// TwinCAT 3 PLC project pruebaPaletizada
// ProgramVersion: 3.1.4024.0
// libraries:
//   Tc2_Standard, * (Beckhoff Automation GmbH)
//   Tc2_System, * (Beckhoff Automation GmbH)
//   Tc3_Module, * (Beckhoff Automation GmbH)
//   VisuSymbols,3.5.10.0,System
// project tree:
//   / GlobalTextList.TcGTLO, PlcTask.TcTTO, Visualization Manager.TcVMO (not stored)
//   GVLs/ GVLvars.TcGVL
//   POUs/ MAIN.TcPOU
//   VISUs/ HMI.TcVIS
// real-time tasks:
//   TASK PlcTask: cycle T#10ms, priority 20, ADS port 350

CONFIGURATION pruebaPaletizada
    RESOURCE PLC ON TwinCAT3
        TASK PlcTask(INTERVAL := T#10ms, PRIORITY := 20);
        PROGRAM MAIN WITH PlcTask : MAIN;
    END_RESOURCE
END_CONFIGURATION

// ---- GVLs/GVLvars.TcGVL
{attribute 'qualified_only'}
VAR_GLOBAL
	// Cuadro
	{attribute 'OPC.UA.DA' := '1'}
	botonStart : BOOL;
	{attribute 'OPC.UA.DA' := '1'}
	botonStop : BOOL;
	{attribute 'OPC.UA.DA' := '1'}
	seta : BOOL; 
	{attribute 'OPC.UA.DA' := '1'}
	botonReset : BOOL;
	{attribute 'OPC.UA.DA' := '1'}
	luzStart : BOOL;
	{attribute 'OPC.UA.DA' := '1'}
	luzStop : BOOL;
	{attribute 'OPC.UA.DA' := '1'}
	luzReset : BOOL;
	{attribute 'OPC.UA.DA' := '1'}
	luzVerde : BOOL;
	{attribute 'OPC.UA.DA' := '1'}
	luzRoja : BOOL;
	{attribute 'OPC.UA.DA' := '1'}
	luzAmarilla : BOOL;
	
	
	// Sensores 
	{attribute 'OPC.UA.DA' := '1'}
	sDifusoCintaMaterial : BOOL;
	{attribute 'OPC.UA.DA' := '1'}
	sEntradaPaletizadorMaterial : BOOL;
	{attribute 'OPC.UA.DA' := '1'}
	sEntradaMesaRotation : BOOL;
	{attribute 'OPC.UA.DA' := '1'}
	sSalidaMesaRotacion : BOOL;
	{attribute 'OPC.UA.DA' := '1'}
	sPostPaletizado : BOOL;
	{attribute 'OPC.UA.DA' := '1'}
	sEntradaPaletEnEstacion : BOOL;
	{attribute 'OPC.UA.DA' := '1'}
	sBasePalet : BOOL ;
	{attribute 'OPC.UA.DA' := '1'}
	numProductosCompletos : INT;
	
	

	// Cintas
	{attribute 'OPC.UA.DA' := '1'}
	cintaEntradaMaterial : BOOL;
	{attribute 'OPC.UA.DA' := '1'}
	cintaInclinadaMaterial : BOOL;
	{attribute 'OPC.UA.DA' := '1'}
	cintaEntradaPalets : BOOL;
	{attribute 'OPC.UA.DA' := '1'}
	cintaSalida : BOOL;
	{attribute 'OPC.UA.DA' := '1'}
	cintaPaletEntradaEstacion : BOOL;
	
	// Mesa Giratoria (Monoestable)
	// Output
	{attribute 'OPC.UA.DA' := '1'}
	turnMesaGiratoria : BOOL;
	{attribute 'OPC.UA.DA' := '1'}
	load : BOOL;
	{attribute 'OPC.UA.DA' := '1'}
	unload : BOOL;
	// Input
	{attribute 'OPC.UA.DA' := '1'}
	frontLimit : BOOL; // Limite frontal de la mesa giratoria
	{attribute 'OPC.UA.DA' := '1'}
	backLimit : BOOL; // Limite trasero de la mesa giratoria
	{attribute 'OPC.UA.DA' := '1'}
	minuminRotation : BOOL; // rotation limit 0
	{attribute 'OPC.UA.DA' := '1'}
	maximunRotation : BOOL; // rotation limit 90
	
	// Paletizador Salidas
	{attribute 'OPC.UA.DA' := '1'}
	pusher : BOOL;
	{attribute 'OPC.UA.DA' := '1'}
	turnFlipper : BOOL;
	{attribute 'OPC.UA.DA' := '1'}
	moveClamper : BOOL;
	{attribute 'OPC.UA.DA' := '1'}
	beltPositive : BOOL;
	{attribute 'OPC.UA.DA' := '1'}
	beltNegative : BOOL;
	{attribute 'OPC.UA.DA' := '1'}
	chainPositive : BOOL;
	{attribute 'OPC.UA.DA' := '1'}
	chainNegative : BOOL;
	{attribute 'OPC.UA.DA' := '1'}
	OpenPlate : BOOL;
	{attribute 'OPC.UA.DA' := '1'}
	elevatorUp : BOOL;
	{attribute 'OPC.UA.DA' := '1'}
	elevatorDown : BOOL;
	{attribute 'OPC.UA.DA' := '1'}
	elevatorToLimit : BOOL;
	
	
	// Paletizador Entradas
	{attribute 'OPC.UA.DA' := '1'}
	clamped : BOOL;
	{attribute 'OPC.UA.DA' := '1'}
	plateLimit : BOOL;
	{attribute 'OPC.UA.DA' := '1'}
	pusherLimit : BOOL;
	{attribute 'OPC.UA.DA' := '1'}
	elevatorMoving : BOOL;
	{attribute 'OPC.UA.DA' := '1'}
	elevatorBackLimit : BOOL;
	{attribute 'OPC.UA.DA' := '1'}
	elevatorFrontLimit : BOOL;
	
	
	

END_VAR

// ---- POUs/MAIN.TcPOU
PROGRAM MAIN
VAR
	enclaveStart: BOOL;
	cintaEntradaMaterial: BOOL;
	cintaInclinadaMaterial: BOOL;
	cintaEntradaPalets: BOOL;
	cintaSalida: BOOL;
	turnPaletizador: BOOL;
	luzVerde: BOOL;
	luzAmarilla : bool;
	luzRoja: BOOL;
	emergencia : bool;
	turnMesaGiratoria: BOOL;
	load: BOOL;
	unload: BOOL;
	pusher: BOOL;
	turnFlipper: BOOL;
	moveClamper: BOOL;
	beltPositive: BOOL;
	beltNegative: BOOL;
	chainPositive: BOOL;
	chainNegative: BOOL;
	openPlate: BOOL;
	elevatorUp: BOOL;
	elevatorDown: BOOL;
	elevatorToLimit: BOOL;
	cintaPaletEntradaEstacion : BOOL;
	contadorVector: INT;
	MatrizElemLista: BOOL;
	PaletListo: bool;
	timerOpenPlate: TON;
	paletizadoListo : bool;
	girando: BOOL;
	flancoEntradaPalets: F_TRIG;
	flancoPusher : R_TRIG;
	flancoPlato: R_TRIG;
	flancoEntradaMaterial : F_TRIG;
	contadorMatriz : int;
	timerAbrirPusher: TOn;
	startTimerPusher: BOOL;
	esperaPusher: BOOL;
	esperaPusher2: BOOL;
	timerVector: ton;
	startTimerVector: BOOL;
	
	recogerPusher: BOOL;
	senalAnterior: INT;
	senalActual: INT;
	pusherLimitAnt: BOOL;
	flancoPusherManual: BOOL;
	clamp: BOOL;
	flancoPlateManual: BOOL;
	plateLimitAnt: BOOL;
	bajandoPalet: BOOL;
	flancoPostPaletizado: F_TRIG;
	flancoMoving : F_TRIG;
	flancoMoVING2 : f_trig;
	paletArriba: BOOL;
	luzStart: BOOL;
	luzStop: BOOL;
	luzReset: BOOL;
	mesaCargada: BOOL;
	girandoMesa: BOOL;
	timerBajadaPalet: TON;
	startTimerPalet: BOOL;
	timerSubidaPalet: TON;
	flancoBasePalet : R_trig;
	saliendo: BOOL;
	numProductosCompletos: INT;
END_VAR

(*
	1 - Boton de start (enclave + cintas emisoras + turn de paletizador)
	
	2 - Boton de stop
	
	3 - Palets
		- detectar palet en mesa de rotacion
		- girar mesa de rotacion (con flanco de bajada de sensor de entrada)
		- arrancar mesa de rotacion y cinta de salida
		- retornar mesa a posicion inicial (flanco sensor salida)
		- colocar palet en base del paletizador
	
	4 - Objeto a paletizar
		- arrancar cinta inclinada con flanco de sensor 
		- activar pusher con 2 objetos (contador por sensor)
		- cuando se hizo push 2 veces (4 objetos sobre plato) -> elevar paletizaodr
		- paletizaodr elevado -> abrir plato con objetos
		- bajar palet cargado 
		- cerrar plato
		- activar cinta para sacar palet cargado de la estacion

*)
luzStart := FALSE;
luzStop := FALSE;
luzReset := FALSE;

IF GVLvars.botonStart AND NOT emergencia THEN
	enclaveStart := TRUE;
	//Arrancar cintas emisoras
	cintaEntradaMaterial := TRUE;
	cintaInclinadaMaterial := TRUE;
	cintaEntradaPalets := TRUE;
	cintaSalida := TRUE;
	turnPaletizador := TRUE;
	luzStart := TRUE;
	luzVerde := TRUE;
	luzAmarilla := FALSE;
	luzRoja := FALSE;
END_IF

IF NOT GVLvars.botonStop AND NOT emergencia THEN
	enclaveStart := FALSE;
	luzStop := TRUE;
	luzVerde := FALSE;
	luzAmarilla := TRUE;
	luzRoja := FALSE;
	cintaEntradaMaterial := FALSE;
	cintaInclinadaMaterial := FALSE;
	cintaEntradaPalets := FALSE;
	cintaPaletEntradaEstacion := FALSE;
	cintaSalida := FALSE;
	turnPaletizador := FALSE;
	turnMesaGiratoria := FALSE ;
	load := FALSE ;
	unload := FALSE;
END_IF

IF NOT GVLvars.seta THEN
	enclaveStart := FALSE;
	luzVerde := FALSE;
	luzAmarilla := FALSE;
	luzRoja := TRUE;
	emergencia := TRUE; 
	cintaEntradaMaterial := FALSE;
	cintaInclinadaMaterial := FALSE;
	cintaEntradaPalets := FALSE;
	cintaPaletEntradaEstacion := FALSE;
	cintaSalida := FALSE;
	turnPaletizador := FALSE;
	//turnMesaGiratoria := FALSE ;
	load := FALSE ;
	unload := FALSE;
END_IF

IF GVLvars.seta AND emergencia THEN
	IF GVLvars.botonReset THEN
		enclaveStart := TRUE;
		luzVerde := TRUE;
		luzAmarilla := FALSE;
		luzRoja := FALSE;
		emergencia := FALSE;
		cintaEntradaMaterial := TRUE;
		cintaInclinadaMaterial := TRUE;
		cintaEntradaPalets := TRUE;
		cintaPaletEntradaEstacion := TRUE;
		cintaSalida := TRUE;
		turnPaletizador := TRUE;
//		turnMesaGiratoria := TRUE ;
//		load := TRUE ;
//		unload := TRUE;
	END_IF
END_IF

	// Si se detecta objeto en la salida de la cinta se activa la inclinada
//	IF  GVLvars.sDifusoCintaMaterial THEN
//		 cintaInclinadaMaterial := TRUE;
//	END_IF


// --------------------------- Material. Parte Superior ---------------------------
IF enclaveStart AND NOT emergencia THEN
	
	flancoEntradaMaterial(CLK:=GVLvars.sEntradaPaletizadorMaterial);
	
	IF  flancoEntradaMaterial.Q THEN
			beltPositive := TRUE;
			contadorVector := contadorVector + 1;
	END_IF

	// Si se dispone de una columna (2 elementos) se empuja hacia el plato
	IF contadorVector >= 2 AND paletListo THEN
		startTimerVector := TRUE;
		
	END_IF
	timerVector(IN := startTimerVector, PT:=T#2S);
		
	IF timerVector.Q THEN
		esperaPusher := TRUE;
		startTimerVector := FALSE;
		cintaEntradaMaterial := FALSE;
		cintaInclinadaMaterial := FALSE;
	END_IF
	
	flancoPusher(CLK:=GVLvars.pusherLimit);
	
	IF esperaPusher THEN
		beltPositive := FALSE;
		pusher := TRUE;
//		cintaEntradaMaterial := FALSE;
//		cintaInclinadaMaterial := FALSE;
		
		//Si el cilindro se extendio de todo (empujo completamente al plato)
		IF flancoPusher.Q THEN
			//startTimerVector:=FALSE;
			pusher := FALSE;
			clamp := TRUE;
			//beltPositive := TRUE;
			contadorVector := 0;
			esperaPusher := FALSE;
			MatrizElemLista := TRUE;
		END_IF
	END_IF
	
	
	



// --------------------------- Palets. Parte Inferior ---------------------------
	flancoEntradaPalets(CLK:=GVLvars.sEntradaMesaRotation);
	IF GVLvars.backLimit  THEN
		load := TRUE;
		mesaCargada := TRUE;
		
		//turnMesaGiratoria := TRUE;
	END_IF
	
	IF mesaCargada THEN
		load:=TRUE;
	END_IF
	
	IF girandoMesa THEN 
		turnMesaGiratoria := TRUE;
	END_IF
//	IF GVLvars.backLimit AND GVLvars.frontLimit THEN
//		load := FA;
		
//	END_IF
	
	// Si llega a la parte frontal de la mesa y todavia no acabo de rotar se paara
	IF GVLvars.frontLimit AND NOT GVLvars.maximunRotation THEN
		load := FALSE;
		turnMesaGiratoria := TRUE;
		girandoMesa := TRUE;
	// Si esta en la parte frontal de la mesa y esta giro completamente
	ELSIF GVLvars.frontLimit AND GVLvars.maximunRotation THEN
		load := TRUE;
		cintaPaletEntradaEstacion := TRUE;
	// Si no hay nada en la parte frontal, mesa girada del todo y ya paso el palet
	// se podrias comprobar solo con el sensor difuso
	ELSIF NOT GVLvars.frontLimit AND GVLvars.maximunRotation AND GVLvars.sSalidaMesaRotacion THEN
		turnMesaGiratoria := FALSE;
		mesaCargada := FALSE;
		girandoMesa := FALSE;
		//ScintaPaletEntradaEstacion := TRUE;
	END_IF

	flancoEntradaPalets(CLK:=GVLvars.sEntradaPaletEnEstacion);
	
	 IF  flancoEntradaPalets.Q THEN 
		 chainPositive := TRUE;
		 saliendo := FALSE;
	 END_IF
	 
	 IF GVLvars.elevatorFrontLimit AND PaletListo = FALSE and saliendo = false THEN
		 chainPositive := FALSE;
		 elevatorToLimit := TRUE;
		 elevatorUp := TRUE;
		 PaletListo := TRUE;
		 elevatorDown := FALSE;
		 openPlate := FALSE; // mieentras no este arriba el palet no se abre el plato
		 
	 END_IF
	 
	 
	 
	 flancoPlato(CLK:=GVLvars.plateLimit);
	 
	// Si el palet esta listo y los elementos agrupados
	IF MatrizElemLista AND PaletListo THEN
		openPlate := TRUE; // Se abre al plato con los materiales
		//timerOpenPlate(IN:=openPlate, PT:= T#2S); // se espera a que este completamente abierto
		// si las compuertas del plato estan completamente abiertas
		IF flancoPlato.Q THEN
			elevatorToLimit := TRUE; // se desactiva la senal de subida del palet
			elevatorUp := FALSE; 
			//paletListo := FALSE;
			elevatorDown := TRUE; //  se activa la senal de bajada
			paletizadoListo := TRUE;
			openPlate := FALSE;
			cintaEntradaMaterial := TRUE;
			cintaInclinadaMaterial := TRUE;
			MatrizElemLista := FALSE;
			
		END_IF
	END_IF
	 flancoBasePalet(CLK:=GVLvars.sBasePalet);
	//timerBajadaPalet(IN:=paletizadoListo, PT:=T#2S);
	// Si el palet esta cargado con los materiales se dirige hacia el remover
	IF flancoBasePalet.Q THEN
		chainPositive := TRUE;
		cintaSalida := TRUE;
		elevatorToLimit := FALSE; // se desactiva la senal de subida del palet
		elevatorUp := FALSE; 
		elevatorDown := FALSE; //  se activa la senal de bajada
		
	END_IF
	
	IF GVLvars.sPostPaletizado THEN
			chainPositive := FALSE;	
			paletizadoListo := FALSE;
			paletListo := FALSE;
			openPlate := FALSE;
			saliendo := TRUE;
			numProductosCompletos := numProductosCompletos + 1;
			
		END_IF	
END_IF
// --------------------------- Actualizar salidas ---------------------------

// Paletizador (salidas)
// Cuadro (salidas)
GVLvars.luzVerde := luzVerde;
GVLvars.luzRoja := luzRoja;
GVLvars.luzAmarilla := luzAmarilla;

// Cintas (salidas)
GVLvars.cintaEntradaMaterial := cintaEntradaMaterial;
GVLvars.cintaInclinadaMaterial := cintaInclinadaMaterial;
GVLvars.cintaEntradaPalets := cintaEntradaPalets;
GVLvars.cintaSalida := cintaSalida;
GVLvars.cintaPaletEntradaEstacion := cintaPaletEntradaEstacion;

// Mesa Giratoria (salidas)
GVLvars.turnMesaGiratoria := turnMesaGiratoria;
GVLvars.load :=  load;
GVLvars.unload := unload;


// Paletizador (salidas)
GVLvars.pusher := pusher;
GVLvars.turnFlipper := turnFlipper;
GVLvars.moveClamper := moveClamper;
GVLvars.beltPositive := beltPositive;
GVLvars.beltNegative := beltNegative;
GVLvars.chainPositive := chainPositive;
GVLvars.chainNegative := chainNegative;
GVLvars.OpenPlate := openPlate;
GVLvars.elevatorUp := elevatorUp;
GVLvars.elevatorDown := elevatorDown;
GVLvars.elevatorToLimit := elevatorToLimit;
GVLvars.numProductosCompletos := numProductosCompletos;

END_PROGRAM

// ---- GlobalTextList.TcGTLO
TEXTLIST GlobalTextList
  658 = ' 90º'
  760 = '%i'
  30 = 'Abrazadera Base'
  360 = 'Abrazadera Tapa'
  548 = 'Base '
  898 = 'Base elevada'
  313 = 'Base Elevada'
  192 = 'Base en Inferior'
  436 = 'Cinta con Bases'
  679 = 'Cinta con las bases y posteriormente producto final'
  348 = 'Cinta con las tapas '
  583 = 'Cinta con Tapas'
  713 = 'Cinta de Salida'
  444 = 'CONTROLES NUMÉRICOS'
  193 = 'Desplegando Brazo Z'
  736 = 'Desplegar Brazo X'
  5 = 'Empuje Plato'
  176 = 'en 90º'
  777 = 'Indicador de mesa giratoria orientada a 90º'
  953 = 'Indicador de mesa giratoria orinetada a 0ª (posicion de reposo)'
  894 = 'Indicador de un palet sobre la mesa giratoria'
  761 = 'Indicador numérico de los elementos que se encuentran sobre el plato del paletizador'
  359 = 'Mesa en 0º'
  512 = 'Mesa en 90º'
  134 = 'MESA GIRATORIA'
  368 = 'Nº  Elem en Plato'
  730 = 'Nº  productos finales'
  98 = 'Nº  Productos Finales'
  718 = 'Nº elem en Plato'
  135 = 'Número de material en plato'
  50 = 'Palet'
  459 = 'Palet en Base'
  194 = 'Palet en Mesa'
  981 = 'PALETIZADOR'
  804 = 'PARTE INFERIOR'
  388 = 'PARTE SUPERIOR'
  393 = 'Plato Abierto'
  97 = 'PRODUCTO FINAL'
  275 = 'Producto Listo '
  389 = 'Reset'
  678 = 'S'
  857 = 'Seta'
  747 = 'Start'
  828 = 'Stop'
  394 = 'Sujeccion de Tapa (Ventosa)'
  426 = 'Sujección Plato'
  464 = 'Y DE ESTADÍSTICA '
END_TEXTLIST

// ---- VISUs/HMI.TcVIS
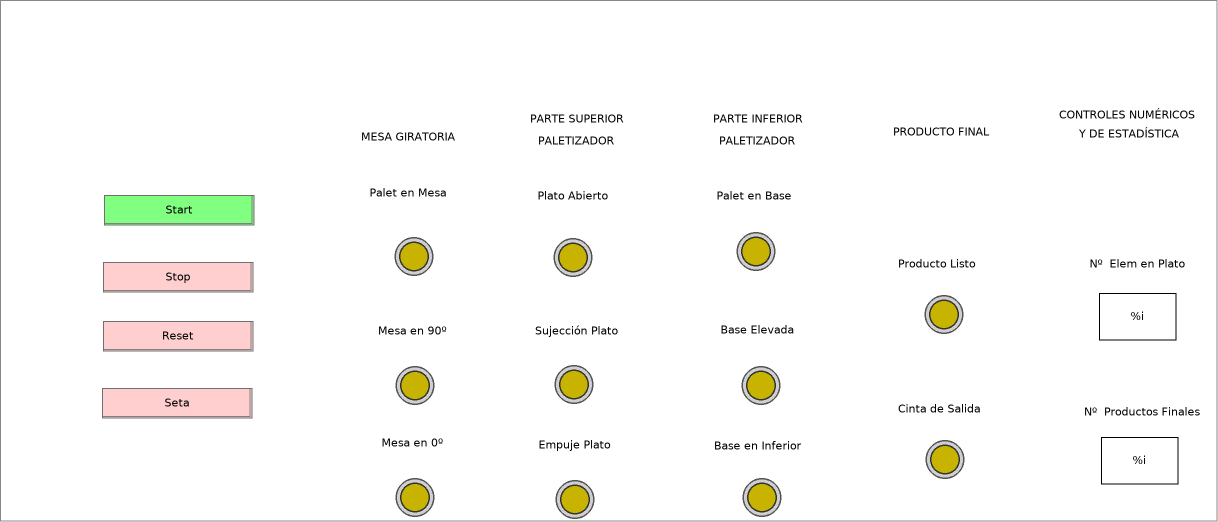
VISUALIZATION HMI  // 1218x522
    Button (104,195 150x30), "Start"
        toggle GVLvars.botonStart
    Button (103,262 150x30), "Stop", colour toggle: NOT GVLvars.botonStop
        toggle GVLvars.botonStop
    Button (103,321 150x30), "Reset", colour toggle: GVLvars.botonReset and MAIN.emergencia
        toggle GVLvars.botonReset
    Button (102,388 150x30), "Seta", colour toggle: Not GVLvars.seta
        toggle GVLvars.seta
    Lamp1 (918,292 52x45), variable: MAIN.paletizadoListo, style: Lamp-Lamp1-Yellow
    Label (890,249 97x30), "Producto Listo"
    Lamp1 (388,234 52x45), tooltip "Indicador de un palet sobre la mesa giratoria", variable: GVLvars.frontLimit, style: Lamp-Lamp1-Yellow
    Label (333,122 150x30), "MESA GIRATORIA"
    Lamp1 (389,363 52x45), tooltip "Indicador de mesa giratoria orientada a 90º", variable: GVLvars.maximunRotation, style: Lamp-Lamp1-Yellow
    Label (371,316 83x30), "Mesa en 90º"
    Label (650,185 190x42)
    Lamp1 (547,235 52x45), tooltip "Cinta con las bases y posteriormente producto final", variable: GVLvars.OpenPlate, style: Lamp-Lamp1-Yellow
    Label (519,175 108x42), "Plato Abierto"
    Lamp1 (548,362 52x45), tooltip "Cinta con las bases y posteriormente producto final", variable: GVLvars.moveClamper, style: Lamp-Lamp1-Yellow
    Label (519,310 115x42), "Sujección Plato"
    Label (333,178 150x30), "Palet en Mesa"
    Lamp1 (389,475 52x45), tooltip "Indicador de mesa giratoria orinetada a 0ª (posicion de reposo)", variable: GVLvars.minuminRotation, style: Lamp-Lamp1-Yellow
    Label (371,428 83x30), "Mesa en 0º"
    Label (502,104 150x30), "PARTE SUPERIOR"
    Label (501,126 150x30), "PALETIZADOR"
    Lamp1 (549,477 52x45), tooltip "Cinta con las bases y posteriormente producto final", variable: GVLvars.pusher, style: Lamp-Lamp1-Yellow
    Label (517,424 115x42), "Empuje Plato"
    Lamp1 (730,229 52x45), tooltip "Cinta con las bases y posteriormente producto final", variable: GVLvars.elevatorFrontLimit, style: Lamp-Lamp1-Yellow
    Label (700,175 108x42), "Palet en Base"
    Lamp1 (735,363 52x45), tooltip "Cinta con las bases y posteriormente producto final", variable: GVLvars.elevatorUp, style: Lamp-Lamp1-Yellow
    Label (700,309 115x42), "Base Elevada"
    Label (683,104 150x30), "PARTE INFERIOR"
    Label (682,126 150x30), "PALETIZADOR"
    Lamp1 (736,475 52x45), tooltip "Cinta con las bases y posteriormente producto final", variable: GVLvars.elevatorDown, style: Lamp-Lamp1-Yellow
    Label (700,425 115x42), "Base en Inferior"
    Label (1036,100 182x30), "CONTROLES NUMÉRICOS"
    Label (1056,119 150x30), "Y DE ESTADÍSTICA"
    Label (866,117 150x30), "PRODUCTO FINAL"
    Lamp1 (919,437 52x45), variable: GVLvars.cintaSalida, style: Lamp-Lamp1-Yellow
    Label (891,394 97x30), "Cinta de Salida"
    Rectangle (1099,293 77x47), "%i", tooltip "Indicador numérico de los elementos que se encuentran sobre el plato del paletizador", text variable: MAIN.contadorVector
    Label (1089,247 97x34), "Nº Elem en Plato"
    Rectangle (1101,437 77x47), "%i", tooltip "Indicador numérico de los elementos que se encuentran sobre el plato del paletizador", text variable: GVLvars.numProductosCompletos
    Label (1076,395 132x34), "Nº Productos Finales"
END_VISUALIZATION
